TYPE Valve :
STRUCT
	bStart : BOOL;
	Output : BOOL;
END_STRUCT
END_TYPE

(* stored: Version 1.1.0.1, ProductVersion 3.1.4024.6
   DUT Valve: Id {72f5a0b7-8ac4-4ebb-903f-ed9260d297ef} *)
